// Mitsubishi GX Works2 project: KhanhHungTap1FX3U   PLC: FX3U/FX3UC

// global labels: Global1
VAR_GLOBAL
  XXLimitN AT M8344 : BOOL;
  XXLimitP AT M8343 : BOOL;
  XXBusy AT M8340 : BOOL;
  XXInterruptInverse AT M8347 : BOOL;
  XXPos AT D8340 : DINT;
  XXAccelTime AT D8348 : INT;
  XXDecelTime AT D8349 : INT;
  XXPosView AT D0 : DINT;
  XXTarPos AT D2 : DINT;
  XXFeed AT D4 : DINT;
  XXTarR AT M0 : BOOL;
  XXTarRSkip AT D6 : INT;
  XXOn AT M1 : BOOL;
  XXRun AT M2 : BOOL;
  XXDirection AT M3 : BOOL;
  XXMinI AT X000 : BOOL;
  XXReadyI AT X004 : BOOL;
  XXPulseO AT Y000 : BOOL;
  XXDirectionO AT Y004 : BOOL;
  XXOnO AT Y002 : BOOL;
  YYLimitN AT M8354 : BOOL;
  YYLimitP AT M8353 : BOOL;
  YYBusy AT M8350 : BOOL;
  YYInterruptInverse AT M8357 : BOOL;
  YYPos AT D8350 : DINT;
  YYAccelTime AT D8358 : INT;
  YYDecelTime AT D8359 : INT;
  YYPosView AT D7 : DINT;
  YYTarPos AT D9 : DINT;
  YYFeed AT D11 : DINT;
  YYTarR AT M4 : BOOL;
  YYTarRSkip AT D13 : INT;
  YYOn AT M5 : BOOL;
  YYRun AT M6 : BOOL;
  YYDirection AT M7 : BOOL;
  YYMinI AT X001 : BOOL;
  YYReadyI AT X005 : BOOL;
  YYPulseO AT Y001 : BOOL;
  YYDirectionO AT Y005 : BOOL;
  YYOnO AT Y003 : BOOL;
  Run AT M8 : BOOL;
  RunI AT X002 : BOOL;
  RunStop AT M9 : BOOL;
  RunStopI AT X003 : BOOL;
  RunState AT D14 : INT;
  RunStateNext AT M10 : BOOL;
  AxisSpinState AT D15 : INT;
  AxisSpinStateNext AT M11 : BOOL;
  AxisTapState AT D16 : INT;
  AxisTapStateNext AT M12 : BOOL;
  FoilExtractState AT D17 : INT;
  FoilExtractStateNext AT M13 : BOOL;
  FoilClampState AT D18 : INT;
  FoilClampStateNext AT M14 : BOOL;
  FoilSupplyState AT D19 : INT;
  FoilSupplyStateNext AT M15 : BOOL;
  FoilExtractTopN AT M16 : BOOL;
  FoilExtractTopNTimer AT TC0 : BOOL;
  FoilExtractTopNTimerDelay AT D20 : INT;
  FoilExtractTopP AT M17 : BOOL;
  FoilExtractTopPTimer AT TC1 : BOOL;
  FoilExtractTopPTimerDelay AT D21 : INT;
  FoilExtractTopPI AT X006 : BOOL;
  FoilExtractTop AT M18 : BOOL;
  FoilExtractTopO AT Y006 : BOOL;
  FoilExtractBotN AT M19 : BOOL;
  FoilExtractBotNTimer AT TC2 : BOOL;
  FoilExtractBotNTimerDelay AT D22 : INT;
  FoilExtractBotP AT M20 : BOOL;
  FoilExtractBotPTimer AT TC3 : BOOL;
  FoilExtractBotPTimerDelay AT D23 : INT;
  FoilExtractBotPI AT X007 : BOOL;
  FoilExtractBot AT M21 : BOOL;
  FoilExtractBotO AT Y007 : BOOL;
  FoilClampN AT M22 : BOOL;
  FoilClampNTimer AT TC4 : BOOL;
  FoilClampNTimerDelay AT D24 : INT;
  FoilClampP AT M23 : BOOL;
  FoilClampPTimer AT TC5 : BOOL;
  FoilClampPTimerDelay AT D25 : INT;
  FoilClampPI AT X010 : BOOL;
  FoilClamp AT M24 : BOOL;
  FoilClampO AT Y010 : BOOL;
  FoilSupplyN AT M25 : BOOL;
  FoilSupplyNTimer AT TC6 : BOOL;
  FoilSupplyNTimerDelay AT D26 : INT;
  FoilSupplyP AT M26 : BOOL;
  FoilSupplyPTimer AT TC7 : BOOL;
  FoilSupplyPTimerDelay AT D27 : INT;
  FoilSupplyPI AT X011 : BOOL;
  FoilSupply AT M27 : BOOL;
  FoilSupplyO AT Y011 : BOOL;
  Overload AT M28 : BOOL;
  OverloadI AT X012 : BOOL;
  OilPump AT M29 : BOOL;
  OilPumpO AT Y012 : BOOL;
  AirBurst AT M30 : BOOL;
  AirBurstO AT Y013 : BOOL;
  AirBurstTimer AT TC8 : BOOL;
  WorkFeedSpin AT D28 : DINT;
  WorkFeedTapDown AT D30 : DINT;
  WorkFeedTapUp AT D32 : DINT;
  FoilFull AT M31 : BOOL;
  FoilFullI AT X013 : BOOL;
  FoilFullTimer AT TC9 : BOOL;
  SpinArray AT D34 : ARRAY [0..5] OF DINT;
  SpinArrayIndex AT D46 : INT;
  SpinTest AT M32 : BOOL;
  SpinTestTimer AT TC10 : BOOL;
  SpinTestTimerDelay AT D47 : INT;
  SettingTapBegin AT D48 : DINT;
  SettingFoilSupplyI AT X014 : BOOL;
  SettingTapSpeed1I AT X015 : BOOL;
  SettingTapSpeed2I AT X016 : BOOL;
  AirReady AT M33 : BOOL;
  AirReadyI AT X017 : BOOL;
  TapCount AT D50 : DINT;
  TapCountAtSupplyEnd AT D52 : DINT;
  StopTap AT M34 : BOOL;
  StopTapTimer AT TC11 : BOOL;
  StopClamp AT M35 : BOOL;
  StopClampPLS AT M36 : BOOL;
  StopClampTimer AT TC12 : BOOL;
  FoilSupplyPTimeoutTimer AT TC13 : BOOL;
  FoilSupplyPTimeoutTimerDelay AT D54 : INT;
END_VAR

// task Task_01 (event TRUE, interval 0, priority 31): POU_01

PROGRAM POU_01
VAR
  fTmp : BOOL;
  fK : DINT;
END_VAR
SET(M8002, M8336);
MOV(M8002, HFFF0, D8336);
RST(M8002, XXInterruptInverse);
RST(M8002, XXOn);
RST(M8002, YYOn);
MOV(M8002, 50, XXAccelTime);
MOV(M8002, 50, XXDecelTime);
MOV(M8002, 150, YYAccelTime);
MOV(M8002, 150, YYDecelTime);
SET(M8002, FoilExtractTop);
SET(M8002, FoilExtractBot);
RST(M8002, SpinTest);
RST(M8002, Overload);
(*1000 pulse = 1 mm, 1 round = 2.0mm, -> servo ppr = 2000*)
DMOV(M8002, 98_304, WorkFeedSpin);
DMOV(M8002, 131_072 / 6, fK);
DMOV(M8002, fK * 0, SpinArray[0]);
DMOV(M8002, fK * 1, SpinArray[1]);
DMOV(M8002, fK * 2, SpinArray[2]);
DMOV(M8002, fK * 3, SpinArray[3]);
DMOV(M8002, fK * 4, SpinArray[4]);
DMOV(M8002, fK * 5, SpinArray[5]);
(*1000 pulse = 1 mm, 1 round = 1.263157mm, -> servo ppr = 1263*)
DMOV(M8002, (1_263 * 2_000) / 60, WorkFeedTapDown);
DMOV(M8002, (1_263 * 2_800) / 60, WorkFeedTapUp);
RST(M8002, TapCount);
DMOV(M8002, 1_000, SettingTapBegin);
(*|||||||||||||||*)
(*|||||||||||||||*)
SET(Run AND RunState = 0 AND AirReady, fTmp);
RST(fTmp, Run);
SET(fTmp, XXOn);
SET(fTmp, YYOn);
RST(fTmp, StopClamp);
SET(fTmp, OilPump);
MOV(fTmp, 1, RunState);
RST(fTmp, fTmp);
SET(RunStop OR Overload, fTmp);
RST(fTmp, Run);
RST(fTmp, RunStop);
RST(fTmp, Overload);
ZRST(fTmp, RunState, FoilSupplyState);
RST(fTmp, XXRun);
RST(fTmp, XXOn);
RST(fTmp, YYRun);
SET(fTmp AND YYOn, StopTap);
SET(fTmp, FoilExtractTop);
SET(fTmp, FoilExtractBot);
RST(fTmp, FoilClamp);
RST(fTmp, FoilSupply);
RST(fTmp, OilPump);
RST(fTmp, fTmp);
OUT_T(StopTap, StopTapTimer, 5);
RST(StopTapTimer, YYOn);
RST(StopTapTimer, StopTap);

(*|||||||||||||||*)
(*|||||||||||||||*)
INC(RunStateNext, RunState);
INC(AxisSpinStateNext, AxisSpinState);
INC(AxisTapStateNext, AxisTapState);
INC(FoilExtractStateNext, FoilExtractState);
INC(FoilClampStateNext, FoilClampState);
INC(FoilSupplyStateNext, FoilSupplyState);
ZRST(M8000, RunStateNext, FoilSupplyStateNext);
DECO(M8000, RunState, 6, M100);
DECO(M8000, AxisSpinState, 6, M200); DECO(M8000, AxisSpinState, 6, M1200); ZRST(NOT XXTarR OR NOT XXReadyI, M1200, M1263);
DECO(M8000, AxisTapState, 6, M300); DECO(M8000, AxisTapState, 6, M1300); ZRST(NOT YYTarR OR NOT YYReadyI, M1300, M1363);
DECO(M8000, FoilExtractState, 6, M400);
DECO(M8000, FoilClampState, 6, M500);
DECO(M8000, FoilSupplyState, 6, M600);
(*|||||||||||||||*)

(*|||||||||||||||*)
(*origin tap, extract, clamp, supply*)
MOV(M101, 1, AxisTapState);
MOV(M101, 1, FoilExtractState);
MOV(M101, 1, FoilClampState);
MOV(M101, 1, FoilSupplyState);
DMOV(M101, TapCount - 4, TapCountAtSupplyEnd);
SET(M101, RunStateNext);
(*origin spin*)
MOV(M102 AND M1320, 1, AxisSpinState);
SET(M102 AND M1320, RunStateNext);
(*ready done, foil supply ready, run command -> cycle start*)
SET(M103 AND M1220 AND M1320 AND M420 AND M520 AND Run, RunStateNext);
(*cycle start*)
SET(M104 AND M1220 AND M1320 AND M420 AND M520, RunStateNext);
(*clamp on*)
MOV(M105, 11, FoilClampState);
RST(M105, XXOn);
SET(M105, RunStateNext);
(*clamp on done -> tap, extract*)
MOV(M106 AND M515, 11, AxisTapState);
MOV(M106 AND M515, 11, FoilExtractState);
SET(M106 AND M515, RunStateNext);
(*tap done -> add tap count, clamp off*)
SET(M107 AND M1320, fTmp);
DINC(fTmp, TapCount);
MOV(fTmp, 16, FoilClampState);
SET(fTmp, RunStateNext);
RST(fTmp, fTmp);
(*clamp off done, extract done -> next hole*)
SET(M108 AND M520 AND M420, fTmp);
MOV(fTmp, 11, AxisSpinState);
SET(fTmp, XXOn);
SET(fTmp, RunStateNext);
RST(fTmp, fTmp);
(*next hole done -> air burst*)
SET(M109 AND M1220, AirBurst);
SET(M109 AND M1220, RunStateNext);
(*return cycle start*)
MOV(M110, 4, RunState);
(*|||||||||||||||*)
(*foil full -> record*)
DMOV(FoilFull, TapCount, TapCountAtSupplyEnd);
(*check*)
SET((TapCount - TapCountAtSupplyEnd) >= 4, fTmp);
RST(NOT SettingFoilSupplyI, fTmp);
MOV(NOT FoilFull AND M620 AND fTmp, 11, FoilSupplyState);
RST(fTmp, fTmp);
(*|||||||||||||||*)

(*|||||||||||||||*)
(*/////get origin spin*)
(*dvit(EN, offset, frequency)*)
DDVIT(M201, 16_384, 32_768, XXPulseO, XXDirection);
SET(M201 AND M8029, AxisSpinStateNext);
RST(M201 AND M8029, M201);
(*reset index and position*)
RST(M1202, SpinArrayIndex);
DMOV(M1202, -fK, XXPos);
MOV(M1202, 20, AxisSpinState);
(*reset index and position*)
RST(M1206, SpinArrayIndex);
DMOV(M1206, -fK, XXPos);
MOV(M1206, 12, AxisSpinState);
(*/////main sequence*)
(*re get origin or next*)
SET(M1211 AND SpinArrayIndex >= 6, fTmp);
MOV(M1211 AND fTmp, 6, AxisSpinState);
SET(M1211 AND NOT fTmp, AxisSpinStateNext);
RST(fTmp, fTmp);
(*move to hole*)
DMOV(M1212, SpinArray[SpinArrayIndex], XXTarPos);
DMOV(M1212, WorkFeedSpin, XXFeed);
INC(M1212, SpinArrayIndex);
SET(M1212, XXRun);
SET(M1212, AxisSpinStateNext);
(*target reach*)
RST(M1213, XXRun);
SET(M1213, AxisSpinStateNext);
(*move to hole done, end*)
SET(M1214, fTmp);
MOV(fTmp, 20, AxisSpinState);
RST(fTmp, fTmp);
(*test*)
OUT_T(M1220 AND SpinTest, SpinTestTimer, SpinTestTimerDelay);
MOV(SpinTestTimer, 11, AxisSpinState);
(*|||||||||||||||*)


(*|||||||||||||||*)
(*/////get origin tap*)
(*at min, jump to move down*)
SET(M301 AND YYMinI, fTmp);
MOV(fTmp, 2, AxisTapState); RST(fTmp, fTmp);
(*not at min, move up*)
SET(M1301 AND NOT YYMinI, fTmp);
RST(fTmp, YYPos);
DMOV(fTmp, -50_000, YYTarPos);
DMOV(fTmp, 5_000, YYFeed);
SET(fTmp, YYRun);
SET(fTmp, AxisTapStateNext); RST(fTmp, fTmp);
(*move up hit limit, reset*)
SET(M302 AND NOT YYBusy, fTmp);
RST(fTmp, YYRun);
RST(fTmp, YYPos);
SET(fTmp, AxisTapStateNext); RST(fTmp, fTmp);
(*move down*)
SET(M1303, fTmp);
DMOV(fTmp, 5_000, YYTarPos);
DMOV(fTmp, 1_000, YYFeed);
SET(fTmp, YYRun);
SET(fTmp, AxisTapStateNext); RST(fTmp, fTmp);
(*move down out min, stop*)
SET(M304 AND NOT YYMinI, fTmp);
RST(fTmp, YYRun);
SET(fTmp, AxisTapStateNext); RST(fTmp, fTmp);
(*stop done, move down xmm*)
SET(M1305, fTmp);
DMOV(fTmp, YYPos + 2_000, YYTarPos);
DMOV(fTmp, 1_000, YYFeed);
SET(fTmp, YYRun);
SET(fTmp, AxisTapStateNext); RST(fTmp, fTmp);
(*move down xmm done -> reset*)
SET(M1306, fTmp);
RST(fTmp, YYPos);
SET(fTmp, AxisTapStateNext); RST(fTmp, fTmp);
(*move to begin*)
DMOV(M1307, SettingTapBegin, YYTarPos);
DMOV(M1307, 5_000, YYFeed);
SET(M1307, YYRun);
SET(M1307, AxisTapStateNext);
(*ready*)
MOV(M1308, 20, AxisTapState);
(*/////main sequence*)
(*move down*)
SET(M1311, fTmp);
DMOV(fTmp, 35_000, YYTarPos);
DMOV(fTmp, WorkFeedTapDown, YYFeed);
SET(fTmp, YYRun);
SET(fTmp, AxisTapStateNext); RST(fTmp, fTmp);
(*target reach or touch max, reset*)
SET(M1312 OR (M312 AND NOT YYBusy), fTmp);
RST(fTmp, YYRun);
SET(fTmp, AxisTapStateNext); RST(fTmp, fTmp);
(*move down done, move up*)
SET(M1313, fTmp);
DMOV(fTmp, SettingTapBegin, YYTarPos);
DMOV(fTmp, WorkFeedTapUp, YYFeed);
SET(fTmp, YYRun);
SET(fTmp, AxisTapStateNext); RST(fTmp, fTmp);
(*move up done, return wait tap hit*)
SET(M1314, fTmp);
MOV(fTmp, 20, AxisTapState); RST(fTmp, fTmp);
(*|||||||||||||||*)

(*|||||||||||||||*)
(*/////get origin foil extract*)
(*top back, bot forward*)
SET(M401, FoilExtractTop);
SET(M401, FoilExtractBot);
SET(M401, FoilExtractStateNext);
(*top back done, bot forward done -> next*)
SET(M402 AND FoilExtractTopP AND FoilExtractBotP, FoilExtractStateNext);
(*end*)
MOV(M403, 20, FoilExtractState);
(*/////main sequence*)
(*top back, bot back*)
RST(M411, FoilExtractTop);
RST(M411, FoilExtractBot);
SET(M411, FoilExtractStateNext);
(*top back done, bot back done -> top forward, bot forward*)
SET(M412 AND FoilExtractTopN, FoilExtractTop);
SET(M412 AND FoilExtractBotN, FoilExtractBot);
SET(M412 AND FoilExtractTopN AND FoilExtractBotN, FoilExtractStateNext);
(*top forwad done, bot forward done -> end*)
MOV(M413 AND FoilExtractBotP AND FoilExtractBotP, 20, FoilExtractState);
(*|||||||||||||||*)

(*|||||||||||||||*)
(*/////get origin foil clamp*)
(*back*)
RST(M501, FoilClamp);
SET(M501, FoilClampStateNext);
(*back done -> next*)
SET(M502 AND FoilClampN, FoilClampStateNext);
(*end*)
MOV(M503, 20, FoilClampState);
(*/////clamp on*)
(*forward*)
SET(M511, FoilClamp);
SET(M511, FoilClampStateNext);
(*forward done -> done*)
MOV(M512 AND FoilClampP, 15, FoilClampState);
(*/////clamp off*)
(*back*)
RST(M516, FoilClamp);
SET(M516, FoilClampStateNext);
(*back done -> done*)
MOV(M517 AND FoilClampN, 20, FoilClampState);
(*|||||||||||||||*)

(*|||||||||||||||*)
(*/////get origin foil supply*)
(*down*)
RST(M601, FoilSupply);
SET(M601, FoilSupplyStateNext);
(*down done -> next*)
SET(M602 AND FoilSupplyN, FoilSupplyStateNext);
(*end*)
MOV(M603, 20, FoilSupplyState);
(*/////supply sequence*)
(*up*)
SET(M611, FoilSupply);
SET(M611, FoilSupplyStateNext);
(*up done -> down*)
RST(M612 AND FoilSupplyP, FoilSupply);
SET(M612 AND FoilSupplyP, FoilSupplyStateNext);
(*down done -> end*)
MOV(M613 AND FoilSupplyN, 20, FoilSupplyState);
(*|||||||||||||||*)

(*|||||||||||||||*)
(*XX*)
RST(XXRun AND XXTarPos = XXPos, XXRun);
DDRVA(XXRun, XXTarPos, XXFeed, XXPulseO, XXDirection);
RST(M8029, XXRun);
OUT(XXDirection, XXDirectionO);
INC(NOT XXRun AND NOT XXBusy AND XXTarRSkip < 5, XXTarRSkip);
RST(XXRun, XXTarRSkip);
OUT(XXTarRSkip >= 5, XXTarR);
(*|||||||||||||||*)
(*YY*)
RST(YYRun AND YYTarPos = YYPos, YYRun);
DDRVA(YYRun, YYTarPos, YYFeed, YYPulseO, YYDirection);
RST(M8029, YYRun);
OUT(NOT YYDirection, YYDirectionO);
INC(NOT YYRun AND NOT YYBusy AND YYTarRSkip < 5, YYTarRSkip);
RST(YYRun, YYTarRSkip);
OUT(YYTarRSkip >= 5, YYTarR);
(**)
OUT(YYMinI, YYLimitN);
(*|||||||||||||||*)

(*|||||||||||||||*)
PLS(RunI, Run); SET(Run, Run);
PLF(RunStopI, RunStop); SET(RunStop, RunStop);
PLF(OverloadI, Overload); SET(Overload, Overload);
OUT_T(NOT RunStopI AND NOT StopClamp, StopClampTimer, 20); SET(StopClampTimer, StopClamp);
SET(StopClamp, FoilClamp);
SET(StopClamp AND FoilClampP, YYOn);
MOV(StopClamp AND FoilClampP, 1, AxisTapState);
RST(StopClamp AND FoilClampP, StopClamp);
RST(StopClamp, RunStop);
(**)
MOV(M8002, 1, FoilExtractTopNTimerDelay);
OUT_T(NOT FoilExtractTop, FoilExtractTopNTimer, FoilExtractTopNTimerDelay); SET(FoilExtractTopNTimer, FoilExtractTopN); RST(FoilExtractTopNTimer, FoilExtractTopP);
MOV(M8002, 2, FoilExtractTopPTimerDelay);
OUT_T(FoilExtractTop, FoilExtractTopPTimer, FoilExtractTopPTimerDelay); SET(FoilExtractTopPTimer, FoilExtractTopP); RST(FoilExtractTopPTimer, FoilExtractTopN);
MOV(M8002, 1, FoilExtractBotNTimerDelay);
OUT_T(NOT FoilExtractBot, FoilExtractBotNTimer, FoilExtractBotNTimerDelay); SET(FoilExtractBotNTimer, FoilExtractBotN); RST(FoilExtractBotNTimer, FoilExtractBotP);
MOV(M8002, 2, FoilExtractBotPTimerDelay);
OUT_T(FoilExtractBot, FoilExtractBotPTimer, FoilExtractBotPTimerDelay); SET(FoilExtractBotPTimer, FoilExtractBotP); RST(FoilExtractBotPTimer, FoilExtractBotN);
(**)
MOV(M8002, 5, FoilClampNTimerDelay);
OUT_T(NOT FoilClamp AND FoilClampPI, FoilClampNTimer, FoilClampNTimerDelay); SET(FoilClampNTimer, FoilClampN); RST(FoilClampNTimer, FoilClampP);
MOV(M8002, 1, FoilClampPTimerDelay);
OUT_T(NOT FoilClampPI, FoilClampPTimer, FoilClampPTimerDelay); SET(FoilClampPTimer, FoilClampP); RST(FoilClampPTimer, FoilClampN);
(**)
MOV(M8002, 10, FoilSupplyNTimerDelay);
OUT_T(NOT FoilSupply, FoilSupplyNTimer, FoilSupplyNTimerDelay); SET(FoilSupplyNTimer, FoilSupplyN); RST(FoilSupplyNTimer, FoilSupplyP);
MOV(M8002, 8, FoilSupplyPTimerDelay);
OUT_T(FoilSupplyPI, FoilSupplyPTimer, FoilSupplyPTimerDelay); SET(FoilSupplyPTimer, FoilSupplyP); RST(FoilSupplyPTimer, FoilSupplyN);
MOV(M8002, 40, FoilSupplyPTimeoutTimerDelay);
OUT_T(FoilSupply, FoilSupplyPTimeoutTimer, FoilSupplyPTimeoutTimerDelay); SET(FoilSupplyPTimeoutTimer, FoilSupplyP); RST(FoilSupplyPTimeoutTimer, FoilSupplyN);
(**)
OUT_T(FoilFullI, FoilFullTimer, 8); OUT(FoilFullTimer, FoilFull);
(*setting feed*)
DMOV(SettingTapSpeed1I, (1263 * 1200) / 60, WorkFeedTapDown);
DMOV(NOT (SettingTapSpeed1I OR SettingTapSpeed2I), (1263 * 1600) / 60, WorkFeedTapDown);
DMOV(SettingTapSpeed2I, (1263 * 2000) / 60, WorkFeedTapDown);
(**)
OUT(AirReadyI, AirReady);
(*|||||||||||||||*)
OUT(XXOn, XXOnO);
OUT(YYOn, YYOnO);
OUT(NOT FoilExtractTop, FoilExtractTopO);
OUT(NOT FoilExtractBot, FoilExtractBotO);
OUT(FoilClamp, FoilClampO);
OUT(FoilSupply, FoilSupplyO);
OUT(OilPump, OilPumpO);
OUT(AirBurst, AirBurstO); OUT_T(AirBurst, AirBurstTimer, 5); RST(AirBurstTimer, AirBurst);
(*|||||||||||||||*)
END_PROGRAM
